	String_1 : STRING; //! First string parameter
	String_2 : STRING; //! Second string parameter
	String_3 : STRING; //! Third string parameter

END_VAR
IF alarms[alarm].bRaised THEN
	RETURN;
END_IF

alarms[alarm].ipArguments.Clear();
IF String_1 <> '' THEN
	alarms[alarm].ipArguments.AddString(String_1);
END_IF

IF String_2 <> '' THEN
	alarms[alarm].ipArguments.AddString(String_2);
END_IF

IF String_3 <> '' THEN
	alarms[alarm].ipArguments.AddString(String_3);
END_IF

alarms[alarm].Raise(USE_DEFAULT_TIMESTAMP);
END_METHOD

END_FUNCTION_BLOCK

// ---- FB_PackML_StateLogger.TcPOU
//! @summary This FB raises events corresponding to <b>state</b> changes within the parent PackML module
FUNCTION_BLOCK FB_PackML_StateLogger
VAR_IN_OUT
    Alarms : ARRAY[1..48] OF FB_TcAlarm; //! Array of alarms for Core PackML events that exist in any PackML enabled module
END_VAR

VAR_INPUT
    ModulePrefix  : STRING;       //! Prefix String for all state change events (Typically the ID and Name of the module in some concatenated form) <TODO> Remove this? </TODO>
    State         : E_PMLState;   //! Current PackML state of the module
    LogAllChanges : BOOL := TRUE; //! If TRUE, all state change events will be logged, regardless of severity, otherwise info alarms are ignored
END_VAR

VAR
    LastState  : E_PMLState := E_PMLState.ePMLState_Aborted; //Saves the previous state each time the block is run
    pTempAlarm : REFERENCE TO FB_TcAlarm;                    //Temporary reference that makes severity checking simpler vs individually checking each change alarm within the case statement
END_VAR

IF State <> LastState THEN //If state has changed
    CASE State OF          //Get the stored alarm that corresponds to the newly entered state and save its reference temporarily
        E_PMLState.ePMLState_Starting:
            pTempAlarm REF= Alarms[E_PackMLBase_Alarms.StateStartingEnter];
        E_PMLState.ePMLState_Execute:
            pTempAlarm REF= Alarms[E_PackMLBase_Alarms.StateExecuteEnter];
        E_PMLState.ePMLState_Completing:
            pTempAlarm REF= Alarms[E_PackMLBase_Alarms.StateCompletingEnter];
        E_PMLState.ePMLState_Complete:
            pTempAlarm REF= Alarms[E_PackMLBase_Alarms.StateCompleteEnter];
        E_PMLState.ePMLState_Resetting:
            pTempAlarm REF= Alarms[E_PackMLBase_Alarms.StateResettingEnter];
        E_PMLState.ePMLState_Idle:
            pTempAlarm REF= Alarms[E_PackMLBase_Alarms.StateIdleEnter];
        E_PMLState.ePMLState_Holding:
            pTempAlarm REF= Alarms[E_PackMLBase_Alarms.StateHoldingEnter];
        E_PMLState.ePMLState_Held:
            pTempAlarm REF= Alarms[E_PackMLBase_Alarms.StateHeldEnter];
        E_PMLState.ePMLState_Unholding:
            pTempAlarm REF= Alarms[E_PackMLBase_Alarms.StateUnholdingEnter];
        E_PMLState.ePMLState_Suspending:
            pTempAlarm REF= Alarms[E_PackMLBase_Alarms.StateSuspendingEnter];
        E_PMLState.ePMLState_Suspended:
            pTempAlarm REF= Alarms[E_PackMLBase_Alarms.StateSuspendedEnter];
        E_PMLState.ePMLState_Unsuspending:
            pTempAlarm REF= Alarms[E_PackMLBase_Alarms.StateUnsuspendingEnter];
        E_PMLState.ePMLState_Stopping:
            pTempAlarm REF= Alarms[E_PackMLBase_Alarms.StateStoppingEnter];
        E_PMLState.ePMLState_Stopped:
            pTempAlarm REF= Alarms[E_PackMLBase_Alarms.StateStoppedEnter];
        E_PMLState.ePMLState_Aborting:
            pTempAlarm REF= Alarms[E_PackMLBase_Alarms.StateAbortingEnter];
        E_PMLState.ePMLState_Aborted:
            pTempAlarm REF= Alarms[E_PackMLBase_Alarms.StateAbortedEnter];
        E_PMLState.ePMLState_Clearing:
            pTempAlarm REF= Alarms[E_PackMLBase_Alarms.StateClearingEnter];
        E_PMLState.ePMLState_Undefined:
            pTempAlarm REF= Alarms[E_PackMLBase_Alarms.StateUndefinedEnter];
    END_CASE

    //If the FB is set to log all changes, log the change, otherwise check the severity of the alarm and log it if it exceeds 'info' severity
    IF LogAllChanges OR (pTempAlarm.eSeverity <> TcEventSeverity.Info AND pTempAlarm.eSeverity <> TcEventSeverity.Verbose) THEN
        pTempAlarm.Raise(0);
    END_IF

    CASE LastState OF //Clear the previous state's event (Events will remain 'Raised' as long as the module remains in that state)
        E_PMLState.ePMLState_Starting:
            Alarms[E_PackMLBase_Alarms.StateStartingEnter].Clear(0, 0);
        E_PMLState.ePMLState_Execute:
            Alarms[E_PackMLBase_Alarms.StateExecuteEnter].Clear(0, 0);
        E_PMLState.ePMLState_Completing:
            Alarms[E_PackMLBase_Alarms.StateCompletingEnter].Clear(0, 0);
        E_PMLState.ePMLState_Complete:
            Alarms[E_PackMLBase_Alarms.StateCompleteEnter].Clear(0, 0);
        E_PMLState.ePMLState_Resetting:
            Alarms[E_PackMLBase_Alarms.StateResettingEnter].Clear(0, 0);
        E_PMLState.ePMLState_Idle:
            Alarms[E_PackMLBase_Alarms.StateIdleEnter].Clear(0, 0);
        E_PMLState.ePMLState_Holding:
            Alarms[E_PackMLBase_Alarms.StateHoldingEnter].Clear(0, 0);
        E_PMLState.ePMLState_Held:
            Alarms[E_PackMLBase_Alarms.StateHeldEnter].Clear(0, 0);
        E_PMLState.ePMLState_Unholding:
            Alarms[E_PackMLBase_Alarms.StateUnholdingEnter].Clear(0, 0);
        E_PMLState.ePMLState_Suspending:
            Alarms[E_PackMLBase_Alarms.StateSuspendingEnter].Clear(0, 0);
        E_PMLState.ePMLState_Suspended:
            Alarms[E_PackMLBase_Alarms.StateSuspendedEnter].Clear(0, 0);
        E_PMLState.ePMLState_Unsuspending:
            Alarms[E_PackMLBase_Alarms.StateUnsuspendingEnter].Clear(0, 0);
        E_PMLState.ePMLState_Stopping:
            Alarms[E_PackMLBase_Alarms.StateStoppingEnter].Clear(0, 0);
        E_PMLState.ePMLState_Stopped:
            Alarms[E_PackMLBase_Alarms.StateStoppedEnter].Clear(0, 0);
        E_PMLState.ePMLState_Aborting:
            Alarms[E_PackMLBase_Alarms.StateAbortingEnter].Clear(0, 0);
        E_PMLState.ePMLState_Aborted:
            Alarms[E_PackMLBase_Alarms.StateAbortedEnter].Clear(0, 0);
        E_PMLState.ePMLState_Clearing:
            Alarms[E_PackMLBase_Alarms.StateClearingEnter].Clear(0, 0);
        E_PMLState.ePMLState_Undefined:
            Alarms[E_PackMLBase_Alarms.StateUndefinedEnter].Clear(0, 0);
    END_CASE

    LastState := State; //Store previous state
END_IF

(*! <description> The current state is compared against the mode during the last call.  The corresponding events are raised/cleared as the state is changed.
<b>This FB is called from FB_PMLModuleBase.StateControl.  Further calls are not necessary.</b></description>*)

END_FUNCTION_BLOCK

// ---- Tests/ModeAndStateTests/T_CantChangeModInExecute.TcPOU
FUNCTION_BLOCK T_CantChangeModInExecute EXTENDS T_UnitTestBase
VAR
  em : EquipmentModule;
  actual, expected : E_PMLUnitMode;
  actualState, expectedState : E_PMLState;
  scanCounter : INT;
  myTestState : (ARRANGE, ACT, ASSERT);
END_VAR

CASE myTestState OF

  ARRANGE:
    em.CyclicLogic();

    IF em.InitComplete THEN
      myTestState := ACT;
      em.ChangeState(E_PMLCommand.ePMLCommand_Clear);
    END_IF

    CycleModuleLogicToAllowChangesToFilterThrough();
    em.ChangeState(E_PMLCommand.ePMLCommand_Reset);

    CycleModuleLogicToAllowChangesToFilterThrough();
    em.ChangeState(E_PMLCommand.ePMLCommand_Start);
    CycleModuleLogicToAllowChangesToFilterThrough();

  ACT:
      
    em.ChangeMode(E_PMLUnitMode.ePMLUnitMode_Maintenance);
    CycleModuleLogicToAllowChangesToFilterThrough();

    actual := em.CurrentMode;
    expected := E_PMLUnitMode.ePMLUnitMode_Production;
    myTestState := ASSERT;
    
    actualState := em.CurrentState;
    expectedState := E_PMLState.ePMLState_Execute;

  ASSERT:
    assertion.AssertEquals_UINT(TO_UINT(expected), TO_UINT(actual), 'actualState := em.CurrentState;');
    assertion.AssertEquals_UINT(TO_UINT(actual), TO_UINT(expected), 'actual := em.CurrentMode');
    myTestState := ARRANGE;
    TestFinished();

END_CASE

METHOD CycleModuleLogicToAllowChangesToFilterThrough : BOOL
VAR_INST
	i: INT;

END_VAR
//em.CyclicLogic();
//CycleModuleLogicToAllowChangesToFilterThrough := i >= 100;
//i := SEL(i >= 100, i + 1, 0);

FOR i := 0 TO 100 DO
  em.CyclicLogic();
END_FOR
END_METHOD

END_FUNCTION_BLOCK

// ---- Tests/ModeAndStateTests/T_JogThroughStates.TcPOU
FUNCTION_BLOCK T_JogThroughStates EXTENDS T_UnitTestBase
VAR
  em : EquipmentModule;
  cmdTriggered : BOOL;
  actual, expected : Tc3_PackML_V2.E_PMLState;
  scanCounter : INT;
  myTestState : (ARRANGE, ACT, ASSERT);
END_VAR


CycleModuleLogicToAllowChangesToFilterThrough();

IF em.InitComplete THEN
  myTestState := ACT;
  em.ChangeState(E_PMLCommand.ePMLCommand_Clear);
END_IF

// clearing -> stopped
CycleModuleLogicToAllowChangesToFilterThrough();
actual := em.CurrentState;
assertion.AssertEquals_UINT(TO_UINT(actual), TO_UINT(E_PMLState.ePMLState_Stopped), 'clearing -> stopped assert : actual := em.CurrentState;');

// stopped -> Idle
em.ChangeState(E_PMLCommand.ePMLCommand_Reset);
CycleModuleLogicToAllowChangesToFilterThrough();
actual := em.CurrentState;
assertion.AssertEquals_UINT(TO_UINT(actual), TO_UINT(E_PMLState.ePMLState_Idle), 'stopped -> Idle assert : actual := em.CurrentState;');

// Idle - > Execute
em.ChangeState(E_PMLCommand.ePMLCommand_Start);
CycleModuleLogicToAllowChangesToFilterThrough();
actual := em.CurrentState;
assertion.AssertEquals_UINT(TO_UINT(actual), TO_UINT(E_PMLState.ePMLState_Execute), 'Idle - > Execute assert : actual := em.CurrentState;');

// Execute -> Hold
em.ChangeState(E_PMLCommand.ePMLCommand_Hold);
CycleModuleLogicToAllowChangesToFilterThrough();
actual := em.CurrentState;
assertion.AssertEquals_UINT(TO_UINT(actual), TO_UINT(E_PMLState.ePMLState_Held), 'Execute -> Hold assert : actual := em.CurrentState;');

// Hold -> Execute
em.ChangeState(E_PMLCommand.ePMLCommand_Unhold);
CycleModuleLogicToAllowChangesToFilterThrough();
actual := em.CurrentState;
assertion.AssertEquals_UINT(TO_UINT(actual), TO_UINT(E_PMLState.ePMLState_Execute), 'Hold -> Execute assert : actual := em.CurrentState;');

// Execute -> Suspend
em.ChangeState(E_PMLCommand.ePMLCommand_Suspend);
CycleModuleLogicToAllowChangesToFilterThrough();
actual := em.CurrentState;
assertion.AssertEquals_UINT(TO_UINT(actual), TO_UINT(E_PMLState.ePMLState_Suspended), 'Execute -> Suspend assert : actual := em.CurrentState;');

// Suspend - > Execute
em.ChangeState(E_PMLCommand.ePMLCommand_Unsuspend);
CycleModuleLogicToAllowChangesToFilterThrough();
actual := em.CurrentState;
assertion.AssertEquals_UINT(TO_UINT(actual), TO_UINT(E_PMLState.ePMLState_Execute), 'Suspend - > Execute assert : actual := em.CurrentState;');

// Execute -> Complete
em.ChangeState(E_PMLCommand.ePMLCommand_Complete);
CycleModuleLogicToAllowChangesToFilterThrough();
actual := em.CurrentState;
assertion.AssertEquals_UINT(TO_UINT(actual), TO_UINT(E_PMLState.ePMLState_Complete), 'Execute -> Complet assert : actual := em.CurrentState;');

// Complete -> Idle
em.ChangeState(E_PMLCommand.ePMLCommand_Reset);
CycleModuleLogicToAllowChangesToFilterThrough();
actual := em.CurrentState;
assertion.AssertEquals_UINT(TO_UINT(actual), TO_UINT(E_PMLState.ePMLState_Idle), 'Complete -> Idle assert : actual := em.CurrentState;');

// Idle -> Stopped
em.ChangeState(E_PMLCommand.ePMLCommand_Stop);
CycleModuleLogicToAllowChangesToFilterThrough();
actual := em.CurrentState;
assertion.AssertEquals_UINT(TO_UINT(actual), TO_UINT(E_PMLState.ePMLState_Stopped), 'Idle -> Stopped assert : actual := em.CurrentState;');

// Stopped -> Idle
em.ChangeState(E_PMLCommand.ePMLCommand_Reset);
CycleModuleLogicToAllowChangesToFilterThrough();
actual := em.CurrentState;
assertion.AssertEquals_UINT(TO_UINT(actual), TO_UINT(E_PMLState.ePMLState_Idle), 'Stopped -> Idle assert : actual := em.CurrentState;');

// Idle -> Abort
em.ChangeState(E_PMLCommand.ePMLCommand_Abort);
CycleModuleLogicToAllowChangesToFilterThrough();
actual := em.CurrentState;
assertion.AssertEquals_UINT(TO_UINT(actual), TO_UINT(E_PMLState.ePMLState_Aborted), 'Idle -> Abort assert : actual := em.CurrentState;');

TestFinished();

METHOD CycleModuleLogicToAllowChangesToFilterThrough : BOOL
VAR_INST
	i: INT;

END_VAR
//em.CyclicLogic();
//CycleModuleLogicToAllowChangesToFilterThrough := i >= 100;
//i := SEL(i >= 100, i + 1, 0);

FOR i := 0 TO 100 DO
  em.CyclicLogic();
END_FOR
END_METHOD

END_FUNCTION_BLOCK

// ---- Tests/ModeAndStateTests/T_CantChangeStateFromIdleToSuspend.TcPOU
FUNCTION_BLOCK T_CantChangeStateFromIdleToSuspend EXTENDS T_UnitTestBase
VAR
  em : EquipmentModule;
  cmdTriggered : BOOL;
  actual, expected : Tc3_PackML_V2.E_PMLState;
  scanCounter : INT;
  myTestState : (ARRANGE, ACT, ASSERT);
END_VAR

CASE myTestState OF
  ARRANGE:
    CycleModuleLogicToAllowChangesToFilterThrough();

    IF em.InitComplete THEN
      em.ChangeState(E_PMLCommand.ePMLCommand_Clear);
      CycleModuleLogicToAllowChangesToFilterThrough();
      em.ChangeState(E_PMLCommand.ePMLCommand_Reset);
      CycleModuleLogicToAllowChangesToFilterThrough();
      myTestState := ACT;
    END_IF

  ACT:
    em.ChangeState(E_PMLCommand.ePMLCommand_Hold);
    CycleModuleLogicToAllowChangesToFilterThrough();
    actual := em.CurrentState;
    myTestState := ASSERT;

  ASSERT:
    assertion.AssertEquals_UINT(TO_UINT(actual), TO_UINT(E_PMLState.ePMLState_Idle), 'actual := em.CurrentState;');
    TestFinished();
END_CASE

METHOD CycleModuleLogicToAllowChangesToFilterThrough : BOOL
VAR_INST
	i: INT;

END_VAR
//em.CyclicLogic();
//CycleModuleLogicToAllowChangesToFilterThrough := i >= 100;
//i := SEL(i >= 100, i + 1, 0);

FOR i := 0 TO 100 DO
  em.CyclicLogic();
END_FOR
END_METHOD

END_FUNCTION_BLOCK

// ---- Tests/ModeManagerTests/T_AddPackModeSetsCorrectly.TcPOU
FUNCTION_BLOCK T_AddPackModeSetsCorrectly EXTENDS T_UnitTestBase
VAR
  mockState : T_MockStateModule;
  modeManager : T_ModeManager(mockState);

  maintenanceMode : T_BaseMode;
  productionMode : T_BaseMode;
  manualMode : T_BaseMode;

  actualMaintenanceMode, actualProdMode, actualManualMode : I_PackMode;
  expectedMaintenanceMode, expectedProdMode, expectedManualMode : I_PackMode;

  maintenanceResult, productionResult, manualResult : BOOL;
END_VAR

//act
modemanager.AddPackModes(productionMode, maintenanceMode, manualMode);

actualMaintenanceMode := modeManager.MaintenanceMode;
actualProdMode := modeManager.ProductionMode;
actualManualMode := modeManager.ManualMode;
expectedMaintenanceMode := maintenanceMode;
expectedProdMode := productionMode;
expectedManualMode := manualMode;

maintenanceResult := actualMaintenanceMode = expectedMaintenanceMode;
productionResult := actualProdMode = expectedProdMode;
manualResult := actualManualMode = expectedManualMode;

//asert
assertion.AssertEquals_BOOL(TRUE, maintenanceResult, 'maintenanceResult := modeManager.MaintenanceMode = maintenanceMode');
assertion.AssertEquals_BOOL(TRUE, productionResult, 'productionResult := modeManager.ProductionMode = productionMode');
assertion.AssertEquals_BOOL(TRUE, manualResult, 'manualResult := modeManager.ManualMode = manualMode');
TestFinished();

END_FUNCTION_BLOCK

// ---- Tests/ModeManagerTests/Mock Objects/T_MockStateModule.TcPOU
FUNCTION_BLOCK T_MockStateModule IMPLEMENTS I_StateModule
VAR_INPUT
  _currentState : UINT;
END_VAR

PROPERTY CurrentState : Tc3_PackML_V2.E_PMLState
GET
CurrentState := _currentState;
END_GET
END_PROPERTY

END_FUNCTION_BLOCK

// ---- Intecre/PackModes/T_BaseMode.TcPOU
FUNCTION_BLOCK T_BaseMode IMPLEMENTS I_PackMode
VAR_INPUT
END_VAR
VAR_OUTPUT
END_VAR
VAR
END_VAR

{warning 'add method implementation '}
METHOD Aborted
END_METHOD

{warning 'add method implementation '}
METHOD Aborting
END_METHOD

{warning 'add method implementation '}
METHOD Clearing
END_METHOD

{warning 'add method implementation '}
METHOD Complete
END_METHOD

{warning 'add method implementation '}
METHOD Completing
END_METHOD

{warning 'add method implementation '}
METHOD Execute
END_METHOD

{warning 'add method implementation '}
METHOD Held
END_METHOD

{warning 'add method implementation '}
METHOD Holding
END_METHOD

{warning 'add method implementation '}
METHOD Idle
END_METHOD

{warning 'add method implementation '}
METHOD Resetting
END_METHOD

{warning 'add method implementation '}
METHOD Starting
END_METHOD

{warning 'add method implementation '}
METHOD Stopped
END_METHOD

{warning 'add method implementation '}
METHOD Stopping
END_METHOD

{warning 'add method implementation '}
METHOD Suspended
END_METHOD

{warning 'add method implementation '}
METHOD Suspending
END_METHOD

{warning 'add method implementation '}
METHOD Unholding
END_METHOD

{warning 'add method implementation '}
METHOD Unsuspending
END_METHOD

END_FUNCTION_BLOCK

// ---- Tests/ModeManagerTests/T_InitModeManagerWithState.TcPOU
FUNCTION_BLOCK T_InitModeManagerWithState EXTENDS T_UnitTestBase
VAR
  stateModule : T_MockStateModule;
  modeManager : T_ModeManager(stateModule);
  
  actual, expected : UINT;
END_VAR

//arrange
stateModule._currentState := 5;

//act

actual := TO_UINT(modeManager._state.CurrentState);
expected := 5;
//assert
assertion.AssertEquals_UDINT(actual, expected , 'actual := modeManager._state');
TestFinished();

END_FUNCTION_BLOCK

// ---- Tests/ModeManagerTests/T_ModeChangeFromProductionToMaintenance.TcPOU
FUNCTION_BLOCK T_ModeChangeFromProductionToMaintenance EXTENDS T_UnitTestBase
VAR
  mockState : T_MockStateModule;
  modeManager : T_ModeManager(mockState);
  expected, actual : UINT;
END_VAR

CycleModuleLogicToAllowChangesToFilterThrough();
modeManager.ChangeMode(E_PMLUnitMode.ePMLUnitMode_Maintenance);
CycleModuleLogicToAllowChangesToFilterThrough();

actual := TO_UINT(modeManager.CurrentMode);
expected := TO_UINT(E_PMLUnitMode.ePMLUnitMode_Maintenance);
assertion.AssertEquals_UINT(expected, actual, 'actual := TO_UINT(modeManager.CurrentMode)');
TestFinished();

METHOD CycleModuleLogicToAllowChangesToFilterThrough : BOOL
VAR_INST
	i: INT;

END_VAR
FOR i := 0 TO 25 DO
  modeManager.CyclicLogic();
END_FOR
END_METHOD

END_FUNCTION_BLOCK

// ---- Tests/ModeManagerTests/T_ModeInitialisedFromInvalidToProduction.TcPOU
FUNCTION_BLOCK T_ModeInitialisedFromInvalidToProduction EXTENDS T_UnitTestBase
VAR
  mockState : T_MockStateModule;
  modeManager : T_ModeManager(mockState);
  expected, actual : UINT;
END_VAR

CycleModuleLogicToAllowChangesToFilterThrough();

expected := TO_UINT(E_PMLUnitMode.ePMLUnitMode_Production);
actual := TO_UINT(modeManager._CurrentMode);
assertion.AssertEquals_UINT(expected, actual, 'actual := modeManager._CurrentMode'); 

TestFinished();

METHOD CycleModuleLogicToAllowChangesToFilterThrough : BOOL
VAR_INST
	i: INT;

END_VAR
FOR i := 0 TO 25 DO
  modeManager.CyclicLogic();
END_FOR
END_METHOD

END_FUNCTION_BLOCK

// ---- Tests/ModeManagerTests/T_AddCustomPackModeSetsCorrectly.TcPOU
FUNCTION_BLOCK T_AddCustomPackModeSetsCorrectly EXTENDS T_UnitTestBase
VAR
  mockState : T_MockStateModule;
  modeManager : T_ModeManager(mockState);

  customMode : T_BaseMode;
  expected, actual : I_PackMode;

  result : BOOL;
END_VAR

modemanager.AddCustomPackMode(0, customMode);
actual := modeManager.CustomPackModes[0];
expected := customMode;
result := actual = expected;
assertion.AssertEquals_BOOL(TRUE, result, 'result := actual = expected;');
TestFinished();

END_FUNCTION_BLOCK

// ---- Tests/CollectionsTests/Components/T_AddComponentAddedToList.TcPOU
FUNCTION_BLOCK T_AddComponentAddedToList EXTENDS T_UnitTestBase
VAR
  list : T_ComponentsCollection;
  newComponent : T_ComponentMock;
  result : BOOL;
END_VAR

result := list.AddComponent(newComponent);

assertion.AssertEquals_BOOL(TRUE, result, 'list.AddComponent(newComponent);');
TestFinished();

END_FUNCTION_BLOCK

// ---- Tests/CollectionsTests/Components/T_AddComponentCompareResultTrue.TcPOU
FUNCTION_BLOCK T_AddComponentCompareResultTrue EXTENDS T_UnitTestBase
VAR
  list : T_ComponentsCollection;
  newComponent : T_ComponentMock;
  actual : I_ComponentBase;
  expected : I_ComponentBase;
  result : BOOL;
END_VAR

list.AddComponent(newComponent);

expected := newComponent;
list.TryGetComponent(0, component => actual);

result := expected = actual;
assertion.AssertEquals_BOOL(TRUE, result, 'result := expected = actual');
TestFinished();

END_FUNCTION_BLOCK

// ---- Tests/CollectionsTests/Components/T_CountReturnsCorrect.TcPOU
FUNCTION_BLOCK T_CountReturnsCorrect EXTENDS T_UnitTestBase
VAR
  list : T_ComponentsCollection;
  newComponent : ARRAY [1..5] OF T_ComponentMock;
  expected, actual : UDINT;
  result : BOOL;
END_VAR

list.AddComponent(newComponent[1]);
list.AddComponent(newComponent[2]);
list.AddComponent(newComponent[3]);
list.AddComponent(newComponent[4]);

expected := 4;
actual := list.Count;

assertion.AssertEquals_UDINT(expected, actual, 'actual := list.Count');
TestFinished();

END_FUNCTION_BLOCK

// ---- Tests/CollectionsTests/Components/T_ClearGroupCountEqualsZeroCompareEqualsFalse.TcPOU
FUNCTION_BLOCK T_ClearGroupCountEqualsZeroCompareEqualsFalse EXTENDS T_UnitTestBase
VAR
  list : T_ComponentsCollection;
  newComponent : ARRAY [1..5] OF T_ComponentMock;
  afterCountActual, afterCountExpected : UDINT;
  beforeCountActual, beforeCountExpected : UDINT;
  beforeActual, beforeExpected : I_ComponentBase;
  afterActual, afterExpected : I_ComponentBase;
 beforeResult, afterResult : BOOL;
END_VAR

// Arrange
list.AddComponent(newComponent[1]);
list.AddComponent(newComponent[2]);
list.AddComponent(newComponent[3]);
list.AddComponent(newComponent[4]);

// first test before running clear
beforeExpected := newComponent[1];
list.TryGetComponent(0, component => beforeActual);
beforeResult := beforeExpected = beforeActual;

Assertion.AssertEquals_BOOL(TRUE, beforeResult, 'item 0 = list.AddComponent()');
Assertion.AssertEquals_UDINT(4, list.Count, 'list.Count = 4');

//Act
list.ClearGroup();

//Assert 
afterExpected := newComponent[1];
list.TryGetComponent(0, component => afterActual);
afterResult := afterExpected <> afterActual;
Assertion.AssertEquals_BOOL(TRUE, beforeResult, 'afterResult := afterExpected <> afterActual;');

afterCountActual := list.Count;
afterCountExpected := 0;
Assertion.AssertEquals_UDINT(afterCountExpected, afterCountActual, 'afterCountActul = 0');

TestFinished();

END_FUNCTION_BLOCK

// ---- Tests/CollectionsTests/Components/T_AddSameComponentTwiceShouldntAdd.TcPOU
FUNCTION_BLOCK T_AddSameComponentTwiceShouldntAdd  EXTENDS T_UnitTestBase
VAR
  list : T_ComponentsCollection;
  newComponent : T_ComponentMock;
  actual : I_ComponentBase;
  expected : I_ComponentBase;
  result : BOOL;
END_VAR

list.AddComponent(newComponent);
result := NOT list.AddComponent(newComponent);

assertion.AssertEquals_BOOL(TRUE, result, 'result := NOT list.AddComponent(newComponent)');
TestFinished();

END_FUNCTION_BLOCK

// ---- Tests/CollectionsTests/Components/T_GetComponentIndexOutOfBoundaryResultsFalse.TcPOU
FUNCTION_BLOCK T_GetComponentIndexOutOfBoundaryResultsFalse EXTENDS T_UnitTestBase
VAR
  list : T_ComponentsCollection;
  newComponent : T_ComponentMock;
  actual : I_ComponentBase;
  expected : I_ComponentBase;
  result, tryGetResultWithinMax, tryGetResultAboveMax : BOOL;
END_VAR

list.AddComponent(newComponent);

tryGetResultWithinMax := NOT list.TryGetComponent(3, component => actual);
tryGetResultAboveMax := NOT list.TryGetComponent(13, component => actual);

result := actual = 0;
assertion.AssertEquals_BOOL(TRUE, result, 'result');
assertion.AssertEquals_BOOL(TRUE, tryGetResultWithinMax, 'tryGetResultWithinMax');
assertion.AssertEquals_BOOL(TRUE, tryGetResultAboveMax, 'tryGetResultAboveMax');
TestFinished();

END_FUNCTION_BLOCK

// ---- Tests/CollectionsTests/Components/T_AddMoreThanSizeOfCollectionFalse.TcPOU
FUNCTION_BLOCK T_AddMoreThanSizeOfCollectionFalse EXTENDS T_UnitTestBase
VAR
  list : T_ComponentsCollection;
  newComponent : ARRAY [1..201] OF T_ComponentMock;
  expected, actual : UDINT;
  result, resultAddOutOfBoundary : BOOL;
  i : UDINT;
END_VAR

FOR i := 1 TO 200 DO
	list.AddComponent(newComponent[i]);
END_FOR

resultAddOutOfBoundary := NOT list.AddComponent(newComponent[201]);

expected := 200;
actual := list.Count;

assertion.AssertEquals_UDINT(expected, actual, 'actual := list.Count');
assertion.AssertEquals_BOOL(TRUE, resultAddOutOfBoundary, 'resultAddOutOfBoundary');
TestFinished();

END_FUNCTION_BLOCK

// ---- Tests/CollectionsTests/Components/T_ComponentsAllowHmiAllowed.TcPOU
FUNCTION_BLOCK T_ComponentsAllowHmiAllowed EXTENDS T_UnitTestBase
VAR
  list : T_ComponentsCollection;
  newComponent, newComponent2 : T_ComponentMock; 
  actual1, actual2 : BOOL;
END_VAR

// Arrange
list.AddComponent(newComponent);
list.AddComponent(newComponent2);

//Act
list.AllowHMIControl();

//Assert
actual1 := newComponent._hmiAllowed;
actual2 := newComponent2._hmiAllowed;

assertion.AssertEquals_BOOL(TRUE, actual1, 'actual1 := newComponent._hmiAllowed;');
assertion.AssertEquals_BOOL(TRUE, actual1, 'actual2 := newComponent2._hmiAllowed;');
TestFinished();

END_FUNCTION_BLOCK

// ---- Tests/CollectionsTests/Module/T_ModuleCollectionOneNotInitialisedAllNotInitialised.TcPOU
FUNCTION_BLOCK T_ModuleCollectionOneNotInitialisedAllNotInitialised EXTENDS T_UnitTestBase
VAR
  list : T_SubModuleCollection;
  newModule, newModule2 : T_SubModuleMock; 
  actual1, actual2 : BOOL;
END_VAR

// Arrange
list.AddModule(newModule);
list.AddModule(newModule2);

//Act
newModule.dontInitialise := TRUE;
list.CyclicLogic();

//Assert
actual1 := NOT list.InitialisedAll;

assertion.AssertEquals_BOOL(TRUE, actual1, 'actual1 := NOT list.InitialisedAll');
TestFinished();

END_FUNCTION_BLOCK

// ---- Tests/CollectionsTests/Module/T_ModuleCollectionAnyErrorReturnErrorTrue.TcPOU
FUNCTION_BLOCK T_ModuleCollectionAnyErrorReturnErrorTrue EXTENDS T_UnitTestBase
VAR
  list : T_SubModuleCollection;
  newModule, newModule2 : T_SubModuleMock; 
  actual1, actual2 : BOOL;
END_VAR

// Arrange
list.AddModule(newModule);
list.AddModule(newModule2);

//Act
list.CyclicLogic();
newModule._error := TRUE;

//Assert
actual1 := list.AnyError;

assertion.AssertEquals_BOOL(TRUE, actual1, 'list.AnyError;');
TestFinished();

END_FUNCTION_BLOCK

// ---- Tests/CollectionsTests/Module/T_ModuleCollectionAllInAskedStateReturnsCorrectResponse.TcPOU
FUNCTION_BLOCK T_ModuleCollectionAllInAskedStateReturnsCorrectResponse EXTENDS T_UnitTestBase
VAR
  list : T_SubModuleCollection;
  newModule, newModule2 : T_SubModuleMock; 
  actual1, actual2 : BOOL;
END_VAR

// Arrange
list.AddModule(newModule);
list.AddModule(newModule2);

//Act
newModule._Currentstate := Tc3_PackML_V2.E_PMLState.ePMLState_Completing;
newModule2._Currentstate := Tc3_PackML_V2.E_PMLState.ePMLState_Completing;

//Assert
actual1 := list.AllInRequestedState(Tc3_PackML_V2.E_PMLState.ePMLState_Completing);

assertion.AssertEquals_BOOL(TRUE, actual1, 'actual1 := list.AllInAskedState(Tc3_PackML_V2.E_PMLState.ePMLState_Completing');
TestFinished();

END_FUNCTION_BLOCK

// ---- Tests/CollectionsTests/Module/T_ModuleCollectionOneIsNotInAskedStateReturnsCorrectResponse.TcPOU
FUNCTION_BLOCK T_ModuleCollectionOneIsNotInAskedStateReturnsCorrectResponse EXTENDS T_UnitTestBase
VAR
  list : T_SubModuleCollection;
  newModule, newModule2 : T_SubModuleMock; 
  actual1, actual2 : BOOL;
END_VAR

// Arrange
list.AddModule(newModule);
list.AddModule(newModule2);

//Act
newModule._Currentstate := Tc3_PackML_V2.E_PMLState.ePMLState_Completing;
newModule2._Currentstate := Tc3_PackML_V2.E_PMLState.ePMLState_Clearing;

//Assert
actual1 := NOT list.AllInRequestedState(Tc3_PackML_V2.E_PMLState.ePMLState_Completing);

assertion.AssertEquals_BOOL(TRUE, actual1, 'actual1 := NOT list.AllInAskedState(Tc3_PackML_V2.E_PMLState.ePMLState_Completing');
TestFinished();

END_FUNCTION_BLOCK

// ---- Tests/CollectionsTests/Module/T_ModuleCollectionAnyInAskedStateReturnsCorrectResponse.TcPOU
FUNCTION_BLOCK T_ModuleCollectionAnyInAskedStateReturnsCorrectResponse EXTENDS T_UnitTestBase
VAR
  list : T_SubModuleCollection;
  newModule, newModule2 : T_SubModuleMock; 
  actual1, actual2 : BOOL;
END_VAR

// Arrange
list.AddModule(newModule);
list.AddModule(newModule2);

//Act
newModule._Currentstate := Tc3_PackML_V2.E_PMLState.ePMLState_Completing;
newModule2._Currentstate := Tc3_PackML_V2.E_PMLState.ePMLState_Holding;

//Assert
actual1 := list.AnyInRequestedState(Tc3_PackML_V2.E_PMLState.ePMLState_Completing);

assertion.AssertEquals_BOOL(TRUE, actual1, 'actual1 := list.AnyInAskedState(Tc3_PackML_V2.E_PMLState.ePMLState_Completing);');
TestFinished();

END_FUNCTION_BLOCK

// ---- Tests/CollectionsTests/Module/T_ModuleCollectionStateResetReturnsCorrectResponse.TcPOU
FUNCTION_BLOCK T_ModuleCollectionStateResetReturnsCorrectResponse EXTENDS T_UnitTestBase
VAR
  list : T_SubModuleCollection;
  newModule, newModule2 : T_SubModuleMock; 
  actual1, actual2 : BOOL;
END_VAR

// Arrange
list.AddModule(newModule);
list.AddModule(newModule2);

//Act
newModule._Currentstate := Tc3_PackML_V2.E_PMLState.ePMLState_Completing;
newModule2._Currentstate := Tc3_PackML_V2.E_PMLState.ePMLState_Complete;

list.StateReset();

//Assert
actual1 := newModule._commandedState = Tc3_PackML_V2.E_PMLCommand.ePMLCommand_Abort;
actual2 := newModule2._commandedState = Tc3_PackML_V2.E_PMLCommand.ePMLCommand_Reset;

assertion.AssertEquals_BOOL(TRUE, actual1, 'actual1 := newModule._commandedState = Tc3_PackML_V2.E_PMLCommand.ePMLCommand_Abort;');
assertion.AssertEquals_BOOL(TRUE, actual2, 'actual2 := newModule2._commandedState = Tc3_PackML_V2.E_PMLCommand.ePMLCommand_Reset;');
TestFinished();

END_FUNCTION_BLOCK

// ---- Example things/T_ExampleModule.TcPOU
FUNCTION_BLOCK T_ExampleModule EXTENDS FB_PackML_BaseModule IMPLEMENTS I_ExampleEquipment

VAR
  
  cartesianRobot : T_ExampleEquipment;

  myProdMode : T_ExampleMOduleProductionMode;
  maintMode : T_ExampleMOduleProductionMode;
  manualMode : T_ExampleMOduleProductionMode;
 
  xAxis : yAxis, zAxis : T_Axis;
  grabber : T_Grabber;
  paramStruct : ST_ExampleParmas;
END_VAR

ComponentsCollection.AddComponent(xAxis);
ComponentsCollection.AddComponent(yAxis);
ComponentsCollection.AddComponent(zAxis);

SubModulesCollection.AddModule(grabber);
cartesianRobot.AddBits(
  xAxis := xAxis.GetRawAxis(),
  yAxis := yAxis,
  zAxis := zAxis,
  grabber := grabber);
  

paramsStruct.xAxis := xAxis;
paramStruct.yAxis := yAxis;
paramStruct.zAxis := zAxis;
paramStruct.grabber := grabber;


myProdMode.init(THIS^);

ModeManager.AddPackModes(myProdMode,maintMode,manualMode);
ModeManager.ChangeMode(E_PMLUnitMode.ePMLUnitMode_Production);

METHOD PUBLIC PickFromStagingArea : BOOL
VAR_INPUT
  orientationOfPick : ST_Orientation;
END_VAR
END_METHOD

END_FUNCTION_BLOCK

// ---- Example things/T_ExampleMOduleProductionMode.TcPOU
FUNCTION_BLOCK T_ExampleMOduleProductionMode EXTENDS T_BaseMode IMPLEMENTS I_PackMode
VAR_INPUT
END_VAR
VAR_OUTPUT
END_VAR
VAR
//  ComponentsCollection : I_ComponentsCollection;
//  xAxis : I_ComponentBase;
  //_modeInterface : I_PackML_BaseModule;
  _specificEquipmentIWantToUse : I_ExampleEquipment;
END_VAR

{warning 'add method implementation '}
METHOD Aborted
END_METHOD

{warning 'add method implementation '}
METHOD Aborting
END_METHOD

{warning 'add method implementation '}
METHOD Clearing
END_METHOD

{warning 'add method implementation '}
METHOD Complete
END_METHOD

{warning 'add method implementation '}
METHOD Completing
END_METHOD

{warning 'add method implementation '}
METHOD Execute
cartesianRobot.PickFromStagingArea();


//THEN OTHER LOGIC
END_METHOD

METHOD GenericInit
VAR_INPUT
  _mode : I_PackML_BaseModule;
END_VAR
// obvs needs more error checking code.

_modeInterface := _mode;
IF NOT __QUERYINTERFACE(_mode, _specificEquipmentIWantToUse) THEN
  ; // ERRROR
END_IF
END_METHOD

{warning 'add method implementation '}
METHOD Held
END_METHOD

{warning 'add method implementation '}
METHOD Holding
END_METHOD

{warning 'add method implementation '}
METHOD Idle
END_METHOD

{warning 'add method implementation '}
METHOD Resetting
END_METHOD

{warning 'add method implementation '}
METHOD Starting
END_METHOD

{warning 'add method implementation '}
METHOD Stopped
END_METHOD

{warning 'add method implementation '}
METHOD Stopping
END_METHOD

{warning 'add method implementation '}
METHOD Suspended
END_METHOD

{warning 'add method implementation '}
METHOD Suspending
END_METHOD

{warning 'add method implementation '}
METHOD Unholding
END_METHOD

{warning 'add method implementation '}
METHOD Unsuspending
END_METHOD

END_FUNCTION_BLOCK

// ---- Intecre/Axis/T_Axis.TcPOU
FUNCTION_BLOCK T_Axis EXTENDS T_NamedBase IMPLEMENTS I_Axis
VAR
END_VAR

END_FUNCTION_BLOCK

// ---- Intecre/Axis/T_AxisComponent.TcPOU
FUNCTION_BLOCK T_AxisComponent EXTENDS FB_ComponentBase IMPLEMENTS I_AxisComponent
VAR
	_axis: I_Axis;
END_VAR

METHOD GenericInitialise
VAR_INPUT
	Axis : I_Axis;
END_VAR
_axis := Axis;
END_METHOD

END_FUNCTION_BLOCK

// ---- Intecre/CartesianRobot/Modes/T_CartesianRobotMaintenanceMode.TcPOU
FUNCTION_BLOCK T_CartesianRobotMaintenanceMode EXTENDS T_NamedBase IMPLEMENTS I_PackMode
VAR
	_cartesianRobot : I_CartesianRobotModule;
END_VAR

METHOD Initialise
VAR_INPUT
	CartesianRobotModule : I_CartesianRobotModule; 
END_VAR
_cartesianRobot := CartesianRobotModule;
END_METHOD

END_FUNCTION_BLOCK

// ---- Intecre/CartesianRobot/Modes/T_CartesianRobotManualMode.TcPOU
FUNCTION_BLOCK T_CartesianRobotManualMode EXTENDS T_NamedBase IMPLEMENTS I_PackMode
VAR
	_cartesianRobot : I_CartesianRobotModule;
END_VAR

METHOD Initialise
VAR_INPUT
	CartesianRobotModule : I_CartesianRobotModule; 
END_VAR
_cartesianRobot := CartesianRobotModule;
END_METHOD

END_FUNCTION_BLOCK

// ---- Intecre/CartesianRobot/Modes/T_CartesianRobotProductionMode.TcPOU
FUNCTION_BLOCK T_CartesianRobotProductionMode EXTENDS T_NamedBase IMPLEMENTS I_PackMode
VAR
	_cartesianRobot : I_CartesianRobotModule;
END_VAR

METHOD Initialise
VAR_INPUT
	CartesianRobotModule : I_CartesianRobotModule; 
END_VAR
_cartesianRobot := CartesianRobotModule;
END_METHOD

END_FUNCTION_BLOCK

// ---- Intecre/CartesianRobot/T_CartesianRobotModule.TcPOU
FUNCTION_BLOCK T_CartesianRobotModule EXTENDS FB_PackML_BaseModule
VAR
	_xAxis, _yAxis, _zAxis : I_Axis;
	_gripper : I_Gripper;
	_cartesianRobot : I_CartesianRobot;
	
	xAxisComponent : T_AxisComponent;
	yAxisComponent : T_AxisComponent;
	zAxisComponent : T_AxisComponent;
	gripperModule : T_GripperModule;
	
	productionMode : T_CartesianRobotProductionMode;
	maintenanceMode : T_CartesianRobotMaintenanceMode;
	manualMode : T_CartesianRobotManualMode;
END_VAR

METHOD GenericInitialise
VAR
	CartesianRobot : I_CartesianRobot;
	xAxis, yAxis, zAxis : I_Axis; 
	Gripper : I_Gripper;
	Cylinder : I_Cylinder;
END_VAR
_xAxis := xAxis;
_yAxis := yAxis;
_zAxis := zAxis;
_gripper := Gripper;
_cartesianRobot := CartesianRobot;

xAxisComponent.GenericInitialise(_xAxis);
yAxisComponent.GenericInitialise(_yAxis);
zAxisComponent.GenericInitialise(_zAxis);
gripperModule.GenericInitialise(gripper, Cylinder);

_cartesianRobot.GenericInitialise(xAxis, yAxis, zAxis, gripper);
productionMode.Initialise(THIS^);
maintenanceMode.Initialise(THIS^);
manualMode.Initialise(THIS^);

ComponentsCollection.AddComponent(xAxisComponent);
ComponentsCollection.AddComponent(yAxisComponent);
ComponentsCollection.AddComponent(zAxisComponent);
SubModulesCollection.AddModule(gripperModule);
END_METHOD

END_FUNCTION_BLOCK

// ---- Intecre/Gripper/T_GripperModule.TcPOU
FUNCTION_BLOCK T_GripperModule EXTENDS FB_PackML_BaseModule IMPLEMENTS I_GripperModule
VAR
	_gripper : I_Gripper;
	_cylinder : I_Cylinder;
	
	cylinderComponent : T_CylinderComponent;
	
	productionMode : T_GripperProductionMode;
	maintenanceMode : T_GripperMaintenanceMode;
	manualMode : T_GripperManualMode;
END_VAR

METHOD GenericInitialise
VAR_INPUT
	Gripper : I_Gripper;
	Cylinder : I_Cylinder;
END_VAR
_gripper := Gripper;
_cylinder := Cylinder;
cylinderComponent.GenericInitialise(_cylinder);

ComponentsCollection.AddComponent(cylinderComponent);
END_METHOD

END_FUNCTION_BLOCK

// ---- Intecre/Cylinder/T_CylinderComponent.TcPOU
FUNCTION_BLOCK T_CylinderComponent EXTENDS FB_ComponentBase
VAR
	_cylinder : I_Cylinder;
END_VAR

METHOD GenericInitialise
VAR_INPUT
	Cylinder : I_Cylinder; 
END_VAR
_cylinder := Cylinder;
END_METHOD

END_FUNCTION_BLOCK

// ---- Intecre/Gripper/Modes/T_GripperProductionMode.TcPOU
FUNCTION_BLOCK T_GripperProductionMode EXTENDS T_NamedBase IMPLEMENTS I_PackMode
VAR
	_gripper : I_GripperModule;
END_VAR

METHOD Initialise
VAR_INPUT
	Gripper : I_GripperModule;
END_VAR
_gripper := Gripper;
END_METHOD

END_FUNCTION_BLOCK

// ---- Intecre/Gripper/Modes/T_GripperMaintenanceMode.TcPOU
FUNCTION_BLOCK T_GripperMaintenanceMode EXTENDS T_NamedBase IMPLEMENTS I_PackMode
VAR
	_gripper : I_GripperModule;
END_VAR

METHOD Initialise
VAR_INPUT
	Gripper : I_GripperModule;
END_VAR
_gripper := Gripper;
END_METHOD

END_FUNCTION_BLOCK

// ---- Intecre/Gripper/Modes/T_GripperManualMode.TcPOU
FUNCTION_BLOCK T_GripperManualMode EXTENDS T_NamedBase IMPLEMENTS I_PackMode
VAR
	_gripper : I_GripperModule;
END_VAR

METHOD Initialise
VAR_INPUT
	Gripper : I_GripperModule;
END_VAR
_gripper := Gripper;
END_METHOD

END_FUNCTION_BLOCK

// ---- Intecre/CartesianRobot/T_CartesianRobot.TcPOU
FUNCTION_BLOCK T_CartesianRobot EXTENDS T_NamedBase
VAR
	_xAxis, _yAxis, _zAxis : I_Axis;
	_gripper : I_Gripper;
END_VAR

METHOD GenericInitialise : BOOL;
VAR_INPUT
	xAxis, yAxis, zAxis : I_Axis;
	gripper : I_Gripper;
END_VAR
IF xAxis = 0 OR yAxis = 0 OR yAxis = 0 OR gripper = 0 THEN
    RETURN;
END_IF

_xAxis := xAxis;
_yAxis := yAxis;
_zAxis := zAxis;
_gripper := gripper;

GenericInitialise := TRUE;
END_METHOD

END_FUNCTION_BLOCK

// ---- Intecre/Gripper/T_Gripper.TcPOU
FUNCTION_BLOCK T_Gripper EXTENDS T_NamedBase IMPLEMENTS I_Gripper
VAR
END_VAR

END_FUNCTION_BLOCK

// ---- Intecre/Cylinder/T_Cylinder.TcPOU
FUNCTION_BLOCK T_Cylinder EXTENDS T_NamedBase IMPLEMENTS I_Cylinder
VAR
END_VAR

END_FUNCTION_BLOCK

// ---- Project Information/F_GetCompany.TcPOU
// This function has been automatically generated from the project information.
{attribute 'signature_flag' := '1073741824'}
{attribute 'TcGenerated'}
{attribute 'no-analysis'}
FUNCTION F_GetCompany : WSTRING
VAR_INPUT
	
END_VAR

F_GetCompany := "Beckhoff Automation LLC";

END_FUNCTION

// ---- Project Information/F_GetTitle.TcPOU
// This function has been automatically generated from the project information.
{attribute 'signature_flag' := '1073741824'}
{attribute 'TcGenerated'}
{attribute 'no-analysis'}
FUNCTION F_GetTitle : WSTRING
VAR_INPUT
	
END_VAR

F_GetTitle := "SPT PackML Base";

END_FUNCTION

// ---- Project Information/F_GetVersion.TcPOU
// This function has been automatically generated from the project information.
{attribute 'signature_flag' := '1073741824'}
{attribute 'TcGenerated'}
{attribute 'no-analysis'}
FUNCTION F_GetVersion : ST_LibVersion
VAR_INPUT
	
END_VAR

F_GetVersion.iMajor := 3;
F_GetVersion.iMinor := 0;
F_GetVersion.iBuild := 3;
F_GetVersion.iRevision := 0;
F_GetVersion.sVersion := '3.0.3';
F_GetVersion.nFlags := 1;

END_FUNCTION

// ---- Tests/AlarmsTests/T_BaseAlarmsClearAlarmIfRaisedCleared.TcPOU
FUNCTION_BLOCK T_BaseAlarmsClearAlarmIfRaisedCleared EXTENDS T_UnitTestBase
VAR
	baseAlarms : T_BaseAlarms;
END_VAR

//Arrange
baseAlarms.RaiseAlarmWithStringParameters(E_BaseAlarms.ComponentError, '','','');

//Act
baseAlarms.ClearAlarmIfRaised(E_BaseAlarms.ComponentError, resetConfirmation := FALSE);

//Assert
Assertion.AssertEquals_BOOL(Expected:= FALSE, Actual := TRUE, 
						VariableName:= 'baseAlarms.ClearAlarmIfRaised(E_BaseAlarms.ComponentError, resetConfirmation := FALSE);' );
TestFinished();

END_FUNCTION_BLOCK

// ---- GlobalTextList.TcGTLO
TEXTLIST GlobalTextList
  685 = '%s'
  680 = 'Abort'
  452 = 'Clear'
  744 = 'Hold'
  347 = 'MACHINE'
  46 = 'Maintenance'
  904 = 'Manual'
  929 = 'Production'
  181 = 'Reset'
  77 = 'Start'
  516 = 'State: %s'
  828 = 'Stop'
  806 = 'Suspend'
  197 = 'Unhold'
  832 = 'Unsuspend'
END_TEXTLIST

// ---- TestUI.TcVIS
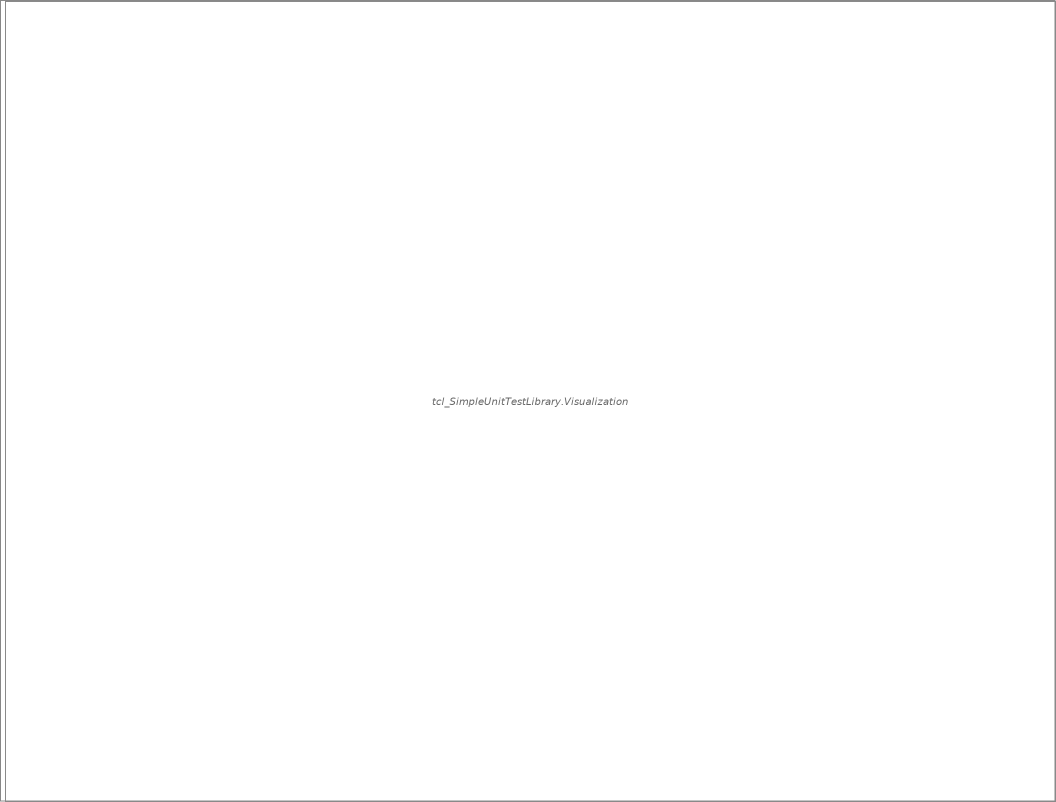
VISUALIZATION TestUI  // 1056x802
    Frame (5,1 1051x801)
        shows tcl_SimpleUnitTestLibrary.Visualization(TestRunner := PRG_Tests.testRunner)
END_VISUALIZATION

// ---- VISUs/V_MachineModule.TcVIS
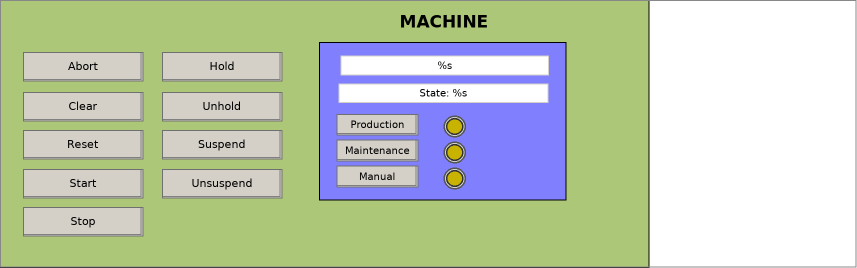
VISUALIZATION V_MachineModule  // 857x268
VAR_IN_OUT
	HMI : ST_PackMLBaseModule_HMI;
END_VAR
    RoundedRectangle (0,0 649x268)
    Button (23,52 120x29), "Abort"
        OnMouseClick: execute { HMI.Command.State := E_PMLCommand.ePMLCommand_Abort; }
    Button (23,92 120x29), "Clear"
        OnMouseClick: execute { HMI.Command.State := E_PMLCommand.ePMLCommand_Clear; }
    Button (23,130 120x29), "Reset"
        OnMouseClick: execute { HMI.Command.State := E_PMLCommand.ePMLCommand_Reset; }
    Button (23,169 120x29), "Start"
        OnMouseClick: execute { HMI.Command.State := E_PMLCommand.ePMLCommand_Start; }
    Button (23,207 120x29), "Stop"
        OnMouseClick: execute { HMI.Command.State := E_PMLCommand.ePMLCommand_Stop; }
    Button (162,52 120x29), "Hold"
        OnMouseClick: execute { HMI.Command.State := E_PMLCommand.ePMLCommand_Hold; }
    Button (162,92 120x29), "Unhold"
        OnMouseClick: execute { HMI.Command.State := E_PMLCommand.ePMLCommand_Unhold; }
    Button (162,130 120x29), "Suspend"
        OnMouseClick: execute { HMI.Command.State := E_PMLCommand.ePMLCommand_Suspend; }
    Button (162,169 120x29), "Unsuspend"
        OnMouseClick: execute { HMI.Command.State := E_PMLCommand.ePMLCommand_Unsuspend; }
    Frame (319,42 247x158)
        shows V_Module(HMI := HMI)
    Label (31,3 826x37), "MACHINE"
END_VISUALIZATION

// ---- VISUs/V_Module.TcVIS
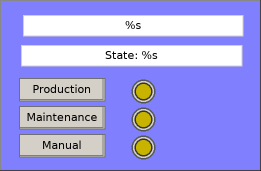
VISUALIZATION V_Module  // 261x171
VAR_IN_OUT
	HMI : ST_PackMLBaseModule_HMI;
END_VAR
    RoundedRectangle (0,0 261x171)
    Textfield (23,15 220x21), "%s", text variable: HMI.Config.Name
    Textfield (21,45 221x21), "State: %s", text variable: HMI.Status.State
    Button (19,78 86x23), "Production"
        OnMouseClick: execute { HMI.Command.Mode := E_PMLUnitMode.ePMLUnitMode_Production; }
    Button (19,106 86x23), "Maintenance"
        OnMouseClick: execute { HMI.Command.Mode := E_PMLUnitMode.ePMLUnitMode_Maintenance; }
    Button (19,134 86x23), "Manual"
        OnMouseClick: execute { HMI.Command.Mode := E_PMLUnitMode.ePMLUnitMode_Manual; }
    Lamp1 (130,78 27x27), variable: HMI.Status.Mode = E_PMLUnitMode.ePMLUnitMode_Production, style: Lamp-Lamp1-Yellow
    Lamp1 (130,106 27x27), variable: HMI.Status.Mode = E_PMLUnitMode.ePMLUnitMode_Maintenance, style: Lamp-Lamp1-Yellow
    Lamp1 (130,134 27x27), variable: HMI.Status.Mode = E_PMLUnitMode.ePMLUnitMode_Manual, style: Lamp-Lamp1-Yellow
END_VISUALIZATION
